// TIA Portal V19 export
TYPE "CTRL_AIN"
   STRUCT
      status : Bool := false;
      sim : "UDT_SIM_REAL";
   END_STRUCT;
END_TYPE
